// TIA Portal V20 export
DATA_BLOCK "LRemoteAccess_Data"   // DB275
TITLE = Data
AUTHOR : Siemens
// Storing data about mobile panel and UCP connection status
// stored: Access Published, MemoryReserve 100
   VAR
      mobilePanel1 : "LRemoteAccess_typeMobilePanel";
      connectionBoxes : Array[1..2] of "LRemoteAccess_typeConnectionBox";
      ActivationMobileDP { S7_SetPoint := 'True'} : "LRemoteAccess_typeMobile_DeActivate";   // Activate Mobile Panel
      DeactivationMobileDP { S7_SetPoint := 'True'} : "LRemoteAccess_typeMobile_DeActivate";   // Deactivate Mobile Panel
      connectionTimeout { S7_SetPoint := 'True'} : Time := T#5S;   // Connection timeout. Keep greater than 3 sec. Default 5 sec.
   END_VAR
BEGIN
   mobilePanel1.connectionTerminated := FALSE;
   mobilePanel1.mpReadBoxID := 0;
   mobilePanel1.mpLifeBit := 5;
   mobilePanel1.mpDesignator := WSTRING#'';
   mobilePanel1.mpKeySwitch := 0;
   mobilePanel1.ucpPointerEnabled := TRUE;
   mobilePanel1.ucpPointerDisabled := FALSE;
   connectionBoxes[1].ID := 18;
   connectionBoxes[2].ID := 19;
   connectionBoxes[1..2].connected := FALSE;
   ActivationMobileDP.Execute := FALSE;
   ActivationMobileDP.RET_VAL := 28672;
   ActivationMobileDP.Busy := FALSE;
   DeactivationMobileDP.Execute := FALSE;
   DeactivationMobileDP.RET_VAL := 28672;
   DeactivationMobileDP.Busy := FALSE;
END_DATA_BLOCK
